(* Schneider Machine Expert - Basic project ECE492_Lab_7_Higginbotham, file version 2.7.0.0 *)
(* ProjectInformations: Name=New project *)

HARDWARE
  Cpu 0: TM221CE16R
  EthernetConfiguration: NetworkName=M221, IpAllocationMode=FixedAddress, IpAddress=192.168.8.202, SubnetMask=255.255.255.0
  SerialLineConfiguration: Baud=Baud19200, Parity=ParityEven, DataBits=DataBits8, StopBits=StopBits1, PhysicalMedium=PhysicalMediumRs485, TransmissionMode=TransmissionModeModbusRtu, SlaveId=1, Addressing=SlaveAddressing
  MastTask: UsePeriodScanMode=false, PeriodScan=100
  FastTask: Period=255
  CpuBehavior: StartingMode=StartAsPreviousState, AutoSaveRamOnEeprom=true, WatchdogPeriod=250

SYMBOLS  (address, symbol, comment, settings)
  %TM0        [Preset=5, Base=OneSecond]
  %IW0.0      [Type=Type_0_10V, Scope=Scope_Normal, Minimum=0, Maximum=1000]

POU New POU
  (* SectionNumber=1 *)

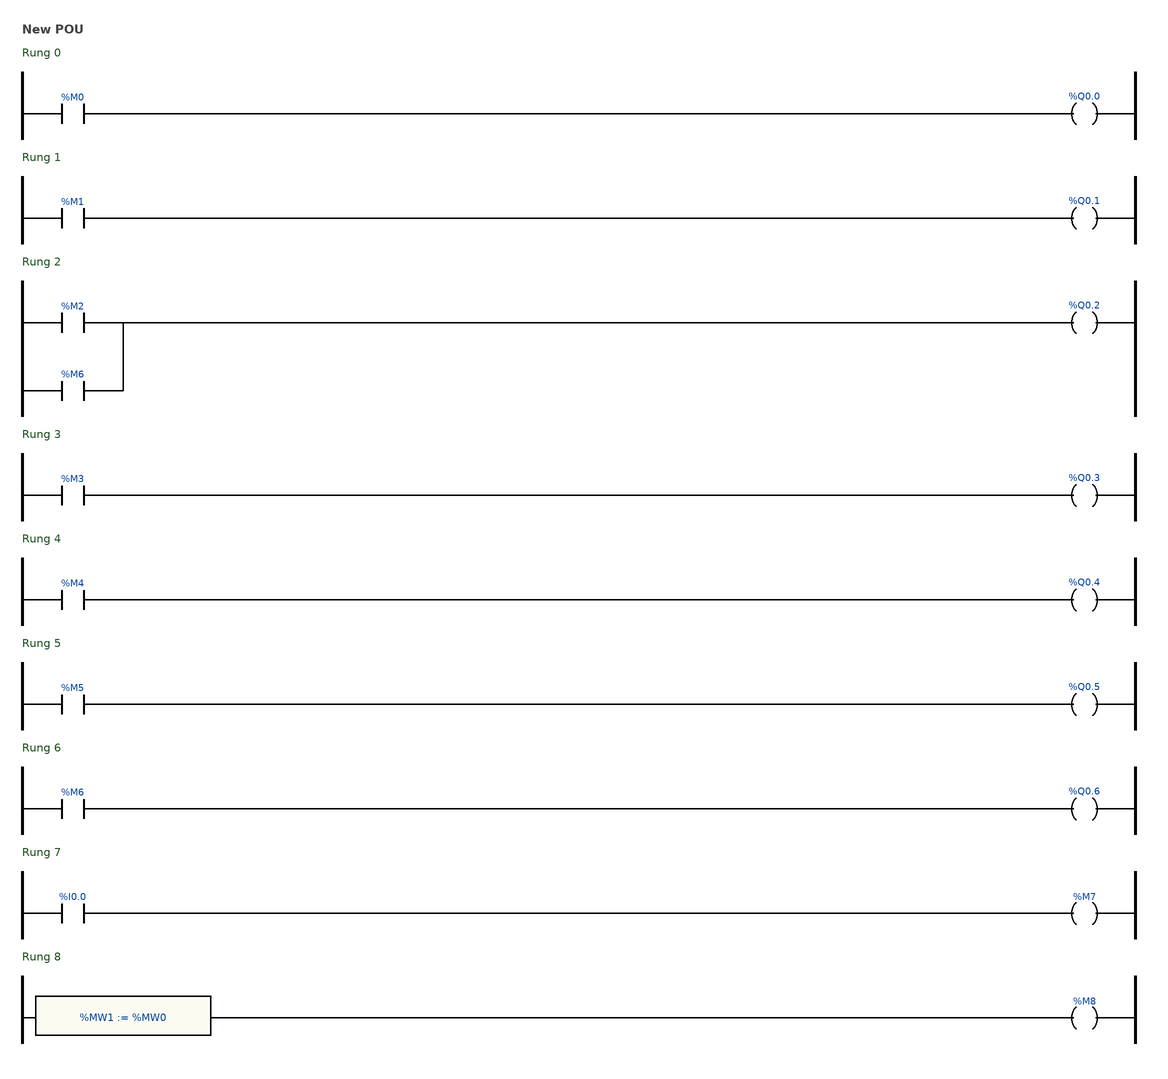

// Rung 0
  LD %M0
  ST %Q0.0
  // as ST:
  //   %Q0.0 := %M0;

// Rung 1
  LD %M1
  ST %Q0.1
  // as ST:
  //   %Q0.1 := %M1;

// Rung 2
  LD %M2
  OR %M6
  ST %Q0.2
  // as ST:
  //   %Q0.2 := %M2 OR %M6;

// Rung 3
  LD %M3
  ST %Q0.3
  // as ST:
  //   %Q0.3 := %M3;

// Rung 4
  LD %M4
  ST %Q0.4
  // as ST:
  //   %Q0.4 := %M4;

// Rung 5
  LD %M5
  ST %Q0.5
  // as ST:
  //   %Q0.5 := %M5;

// Rung 6
  LD %M6
  ST %Q0.6
  // as ST:
  //   %Q0.6 := %M6;

// Rung 7
  LD %I0.0
  ST %M7
  // as ST:
  //   %M7 := %I0.0;

// Rung 8
  LD 1
  OPER [ %MW1 := %MW0 ]
  ST %M8
  // as ST:
  //   %MW1 := %MW0;
  //   %M8 := TRUE;

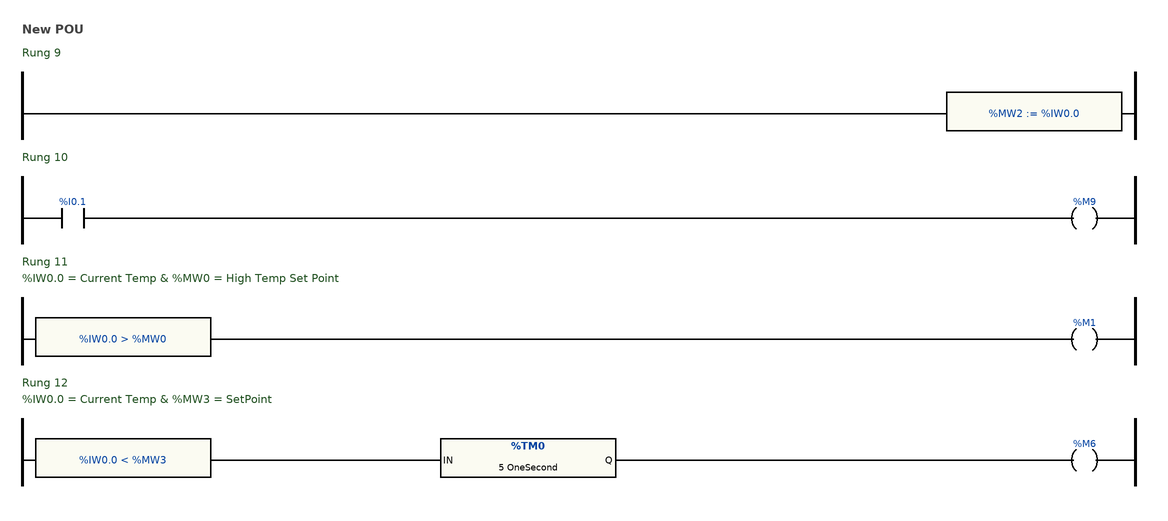

// Rung 9
  LD 1
  [ %MW2 := %IW0.0 ]
  // as ST:
  //   %MW2 := %IW0.0;

// Rung 10
  LD %I0.1
  ST %M9
  // as ST:
  //   %M9 := %I0.1;

// Rung 11
// %IW0.0 = Current Temp & %MW0 = High Temp Set Point
  LD [ %IW0.0 > %MW0 ]
  ST %M1
  // as ST:
  //   %M1 := %IW0.0 > %MW0;

// Rung 12
// %IW0.0 = Current Temp & %MW3 = SetPoint
  BLK %TM0
  LD [ %IW0.0 < %MW3 ]
  IN
  OUT_BLK
  LD Q
  ST %M6
  END_BLK
  // as ST:
  //   %TM0(IN := %IW0.0 < %MW3);
  //   %M6 := %TM0.Q;
